PROGRAM MAIN
VAR	
	/// private var's
	ii						: INT;
	wsClearText				: WSTRING(255);		// clear text for debug
	nOnlineChangesMirror	: UDINT;			// online change tracker
	bInit					: BOOL; 			// PLC init flag
	bRunUnitTest			: BOOL;				// UnitTest
	
	nHmiSize				: ARRAY[0..15] OF UDINT;
END_VAR

///
/// MAIN program - starting point of the PLC project.
/// TP/www.rmth.at/5.2025
/// 

///
/// CHANGES
/// - NAME/DATE/COMMENT

wsClearText := "Run system provider (get time, logger, system and PLC info, ...)";
P_System();

wsClearText := "Init PLC";
M_ChangeWatchdog();

IF NOT M_Init() THEN
	RETURN;
END_IF

wsClearText := "P_Safety";
P_Safety();
	
wsClearText := "Call HMI Controller component";
P_HMI_Controller();

wsClearText := "Call P_Plant";
P_Plant();

wsClearText := "P_Supervision";
P_Supervision(stIO_Cabinet := IO.stControlCabinetIO, nLogger := Services.ILog);

wsClearText := "P_SysSrv";
P_SysSrv();
	
wsClearText := "Run unit tests";
IF bRunUnitTest THEN
	P_UnitTest();
END_IF

Services.b1stShot := FALSE;
Services.bPlcInitDone := TRUE;


(*// DEBUG / TESTS
nHmiSize[0] := SIZEOF(HMI.stHmiInOut);

nHmiSize[1] := SIZEOF(HMI.stHmiTc3);
nHmiSize[2] := SIZEOF(HMI.stHmiTc3.stIn);
nHmiSize[3] := SIZEOF(HMI.stHmiTc3.stOut);

nHmiSize[4] := SIZEOF(HMI.stHmiTc3.stOut.stHeader);
nHmiSize[5] := SIZEOF(HMI.stHmiTc3.stOut.stPopup);
nHmiSize[6] := SIZEOF(HMI.stHmiTc3.stOut.stCounter);
nHmiSize[7] := SIZEOF(HMI.stHmiTc3.stOut.stControlCounter);
nHmiSize[8] := SIZEOF(HMI.stHmiTc3.stOut.stNotificationControl);
nHmiSize[9] := SIZEOF(HMI.stHmiTc3.stOut.stNotificationList);
nHmiSize[10] := SIZEOF(HMI.stHmiTc3.stOut.stNotificationArchiv);
nHmiSize[11] := SIZEOF(HMI.stHmiTc3.stOut.stConditionMonitoring);
nHmiSize[12] := SIZEOF(HMI.stHmiTc3.stOut.stSetupPlant);
nHmiSize[13] := SIZEOF(HMI.stHmiTc3.stOut.stEmergencyStop);
nHmiSize[14] := SIZEOF(HMI.stHmiTc3.stOut.stDoor);
//nHmiSize[15] := SIZEOF(HMI.stHmiTc3.stOut.astStation); *)

ACTION Info:
(*
//----------------------------------------------------------------------

Vorgabe 12.0 s / Stück

Ergebnissdaten Prüflinge: 	iO; Lfd.Nr.;
							
Koordinatensystem Anlage
X = von links nach rechts (Ansicht Vorne)
Y = Vorne (Eingabe) nach hinten
Z = Vertikal						

Stationsauswahl

ST001 Eingabe

----------------------------------------
Schutzbereiche

Schutzbereich 1 -> 	Modul 1 gesamt

//---------------------------------------------------------------------
Anzahl Rund Takt Tisch (RTT) Nestplätze 4 Nester 1

//---------------------------------------------------------------------
Abkürzungen Fehler:
HS = Hochspannung

	
//---------------------------------------------------------------------
pragmas

{text 'todo remove after commissioning'} 
{info 'todo remove after commissioning'} 
{warning 'todo remove after commissioning'} 
{error 'todo remove after commissioning'} 

//----------------------------------------------------------------------

Die wichtigsten Infos zu TC3/RMTH Standard:
	*** min/max und default Werte von Datentypen ***
		RmthTc3Library -> StaticsConstant
		
	*** Stringfunktionen aus RmthTc3Library ***
		aSClearText[EN] := Concat2-10('Text... / ConcatArray(...
		F_RealToString / F_RealToStringEx / F_LRealToString / F_LRealToStringEx
		
	*** Background -> UnitTest ***
		Komponenten hier testen!!!
		
	*** Automatic Sequence Demo ***
		siehe Background -> UnitTest -> TestCases -> StationTest -> FB_TestStation (zb.: DEMO oder M_Sequence)
		
	*** aktuelle PLC System Info ***
		Statics.stPlcSystemInfo
	
--- TC3 Allgemein ---

	*** DATENTYPEN 	***
		https://infosys.beckhoff.com/content/1031/tcplccontrol/html/tcplcctrl_plc_data_types_overview.htm?id=7365416610509907248
	
	*** ATTRIBUTE 	***
		https://infosys.beckhoff.com/content/1031/tc3_plc_intro/54043195664658571.html?id=1095976264130046106
		
	 - Attribut monitoring (Property-OnlineView)
		{attribute 'monitoring' := 'variable'}
		{attribute 'monitoring' := 'call'}
		
		variable: 	Eine implizite Variablen wird angelegt, deren Wert aktualisiert wird, wenn die Applikation die Set oder Get Methode der Eigenschaft aufruft.
		call: 		Der Monitoring-Dienst ruft die Get Methode der Eigenschaft auf
		
		Beispiel:
		{attribute 'monitoring' := 'call'}
		PROPERTY TestState : E_TestCaseState
		
	 - Attribut pack_mode (ändern des Alignments)
		0	aligned, d.h. es treten keine Speicherlücken auf
		1	1-byte-aligned (identisch zu aligned)
		2	2-byte-aligned, d.h. die maximale Größe einer Speicherlücke ist 1 byte
		4	4-byte-aligned, d.h. die maximale Größe einer Speicherlücke ist 3 byte
		8	8-byte-aligned, d.h. die maximale Größe einer Speicherlücke ist 7 byte
		
		Beispiel:
		{attribute 'pack_mode' := '1'}
		TYPE ST_MyStruct:
		
--- Text ---		
		F_CreateDynText("velooffsetchain",0)
		
------------------------------------------------------------------------------------------------------------------------
how to use popup
		
CASE nTestStep OF
	
	0:
		;
	
	10:
		IF fbHmiHandler.M_PopupCheck(E_Popup.ePopup01) THEN
			CASE fbHmiHandler.M_PopupSet(E_Popup.ePopup01,F_CreateDynText("Wasch Prozess Starten ?",0),F_CreateDynText("yes",0),F_CreateDynText("no",0),F_CreateDynText("Info",0),F_CreateDynText("Abbrechen",0)) OF
				1:
					nTestStep :=100;
				2:
					nTestStep :=0;		
				4:	
					nTestStep :=200;
			END_CASE			
		END_IF
	100:
		IF fbHmiHandler.M_PopupCheck(E_Popup.ePopup02) THEN
			CASE fbHmiHandler.M_PopupSet(E_Popup.ePopup02,F_CreateDynText("Wollen Sie wirklich den Wasch Prozess Starten ?? Sicher ??",0),F_CreateDynText("yes",0),F_CreateDynText("",0),F_CreateDynText("Abbruch",0),F_CreateDynText("",0)) OF

				1:
					nTestStep :=200;		
				3:	
					nTestStep :=0;
			END_CASE			
		END_IF
		
	200:
		IF fbHmiHandler.M_PopupCheck(E_Popup.ePopup01) THEN
			CASE fbHmiHandler.M_PopupSet(E_Popup.ePopup01,F_CreateDynText("Prozess Fertig",0),F_CreateDynText("OK",0),F_CreateDynText("",0),F_CreateDynText("",0),F_CreateDynText("",0)) OF
				1:
					nTestStep :=0;
			END_CASE			
		END_IF	
END_CASE

IF FALSE THEN
	IF fbHmiHandler.M_PopupCheck(E_Popup.ePopupSafetyEs) THEN
		fbHmiHandler.M_PopupSet(E_Popup.ePopupSafetyEs,F_CreateDynText("Nothalt nicht OK -> Bitte Quittieren !",0),F_CreateDynText("",0),F_CreateDynText("",0),F_CreateDynText("",0),F_CreateDynText("OK",0)) ;
	END_IF	
END_IF		
		
		
*)
END_ACTION

METHOD PRIVATE M_ChangeWatchdog : BOOL
VAR
END_VAR
wsClearText := "Run onlineChange watchdog";

stPlcAppSystemInfo := Statics.stPlcSystemInfo.stPlcAppSystemInfo;
IF nOnlineChangesMirror <> stPlcAppSystemInfo.OnlineChangeCnt THEN
	wsClearText := "OnlineChange detected -> ReInit!";
	bInit := FALSE;	
	nOnlineChangesMirror := stPlcAppSystemInfo.OnlineChangeCnt;
END_IF
END_METHOD

METHOD PRIVATE M_Init : BOOL
VAR
	// local temp var's
	ISt : IStation;
END_VAR
///
///	PLC INIT: Initialisierung aller Komponenten
/// - Einstellungen treffen
/// - setzen von Referenzen
/// - wichtig: in einem Zyklus fertig!

wsClearText := "Check PLC init done";
IF bInit THEN
	M_Init := TRUE;
	RETURN;
END_IF

wsClearText := "PLC init: first shot setup";
IF Statics.stPlcSystemInfo.stPlcTaskSystemInfo.FirstCycle THEN
	;//P_HMI.recipeManagement.M_ReadRecipe();
END_IF

wsClearText := "PLC init: wait for valid system Time";
IF Statics.dtNow = dtMinValue THEN
	RETURN;
END_IF

{region "configuration and logging"}
wsClearText := "PLC init: setup/load configuration";
stConfig.stLogConfig.eLoggingProvider := E_LoggingProvider.eLoggingProviderFile;
stConfig.stLogConfig.sLogName := 'PlcLog.txt';
stConfig.stLogConfig.sLogPath := '/home/';
stConfig.stLogConfig.eLogLevel := E_LogLevel.eLogLevel_info;

wsClearText := "Set up logging provider";
P_System.fbFileLog.Source := stConfig.stLogConfig.sLogName;
P_System.fbFileLog.sPath := stConfig.stLogConfig.sLogPath;
P_System.fbFileLog.LogLevel := stConfig.stLogConfig.eLogLevel;
	
P_System.fbEventLog.Source := stConfig.stLogConfig.sLogName;
P_System.fbEventLog.LogLevel := stConfig.stLogConfig.eLogLevel;
	
P_System.fbDebugLog.Source := stConfig.stLogConfig.sLogName;
P_System.fbDebugLog.LogLevel := stConfig.stLogConfig.eLogLevel;
IF stConfig.stLogConfig.eLoggingProvider = E_LoggingProvider.eLoggingProviderFile THEN
	Services.ILog := P_System.fbFileLog;
ELSIF stConfig.stLogConfig.eLoggingProvider = E_LoggingProvider.eLoggingProviderEventLog THEN
	Services.ILog := P_System.fbEventLog;
ELSE // default
	Services.ILog := P_System.fbDebugLog;
END_IF

Services.fbEventHandler.Init();

{endregion}

{region "initialize HMI controller and provider"}
wsClearText := "Initialize HMI";
P_HMI_Controller.M_Init();
HMI.fbHmiHwProvider.M_Init();
HMI.fbHmiTc3Provider.M_Init();
{endregion}

{region "initialize components, stations and modules"}

wsClearText := "Initialize plant components";
// plant component initialization here...
	 

wsClearText := "Initialize stations, modules and plant";

// sample 1: quick, default IOs and services:
//		fbSt010OvenA.M_Init();
	 
// sample 2: using custom settings, IOs and services:
//		fbSt010OvenA.Station := E_Station.eStation_ST010_OvenA;
//		fbSt010OvenA.Name := stTextListGlobal.stText_ST010_Name;
//		fbSt010OvenA.Active := TRUE;
//		fbSt010OvenA.Enable := TRUE;
//		fbSt010OvenA.M_SetReferences(IO.st010_OvenA_IO);
//		ISt := fbSt010OvenA.M_InitEx(Services.ILog, Services.fbNotiHandler);
//		fbModul001.M_RegisterStation(ISt);
	 
fbSt010OvenA.M_Init();
fbSt020OvenB.M_Init();
fbSt030Handling.M_Init();
fbSt040Storage.M_Init();
fbSt050Mould.M_Init();
fbModul001.M_Init();
P_Plant.M_Init();

{endregion}

wsClearText := "Initialize Safety";
P_Safety.M_Init();

wsClearText := "Initialize Supervision";
P_Supervision.M_Init();

wsClearText := "PLC init done.";
Services.ILog.AddLog(TO_STRING(wsClearText), sSource, E_LogLevel.eLogLevel_info);

bInit := TRUE;
M_Init := bInit;
END_METHOD

 {attribute 'call_after_online_change_slot' := '1'}
METHOD M_OnlineChange : BOOL
VAR_INPUT
END_VAR
bInit := FALSE;
END_METHOD

END_PROGRAM

(* stored: Version 1.1.0.1
   POU MAIN: Id {bd2e5e27-e7c9-44f5-9dc8-02ae4a0ea03d}, SpecialFunc None
   Action Info: Id {7650a567-0d90-49b9-8119-207eb69b5acf}
   Method M_ChangeWatchdog: Id {33892116-16d7-4e1a-88a7-e35e1857f998}
   Method M_Init: Id {f74952ec-f0a4-4874-996f-0f42b6a228da}
   Method M_OnlineChange: Id {8a450ade-d4bb-4acb-9891-b22f5760d414} *)
